// Struct contains all data from other tasks and controller used for slave control
TYPE ST_SetupInputDataPool :
STRUCT
				
	// UI information, import from UI controller
	m_UIData AT %I*:ST_SlaveUIData;
	
	// safety information, import from safety check task
	m_safetyData AT %I*: ST_SafetyData;
	
	// cart information, import from other task
	m_cartStatus AT %I*:ST_CartStatus;
	
	// slave gravity
	m_setupJnt3Gravity AT %I* : LREAL;
	m_setupJnt5Gravity AT %I* : LREAL;
	
	
END_STRUCT
END_TYPE

(* stored: Version 1.1.0.1, ProductVersion 3.1.4024.12
   DUT ST_SetupInputDataPool: Id {b34d09b2-0ba9-48c6-ad2b-bb4df07793ad} *)
